TYPE "StaProcessData"
VERSION : 0.1
   STRUCT
      Reserved0 : Bool;
      Reserved1 : Bool;
      PartResult : Byte;
      PalletNo : Int;
      Mode : Int;
      PartID : String[48];
      "P-SubPartID" : Array[1..10] of String[48];
   END_STRUCT;

END_TYPE

